// SIMATIC STEP 7 (V5.x) project S7Interface
// CPU: CPU 317-2 PN/DP
// station: Hardware
// station: SIMATIC 300(1)
// station: P_ADR_BUS
// program: Programma S7(1)

SYMBOL_TABLE
"TEST"	DB 1	DB 1
"FETCH"	DB 10	DB 10
"WRITE"	DB 11	DB 11
"FW_TCP"	FB 210	FB 210	// Fetch/Write via TCP
END_SYMBOL_TABLE

// FB 210: know-how protected block, not included

DATA_BLOCK "TEST"	// DB 1
VERSION : 0.1
  STRUCT
   TestBYTE : ARRAY  [0 .. 128 ] OF BYTE ;
   TestCHAR : ARRAY  [0 .. 128 ] OF CHAR ;
   TestWORD : ARRAY  [0 .. 1024 ] OF WORD ;
   TestINT : ARRAY  [0 .. 1024 ] OF INT ;
   TestDWORD : ARRAY  [0 .. 1024 ] OF BOOL ;
   TestDINT : ARRAY  [0 .. 1024 ] OF BOOL ;
   TestBOOL : ARRAY  [0 .. 1024 ] OF BOOL ;
   TestREAL : ARRAY  [0 .. 1024 ] OF REAL ;
   TestSTRING : ARRAY  [0 .. 1024 ] OF STRING  [16 ];
   TestTIME : ARRAY  [0 .. 512 ] OF TIME ;
   TestTOD : ARRAY  [0 .. 512 ] OF TIME_OF_DAY ;
   TestDT : ARRAY  [0 .. 128 ] OF DATE_AND_TIME ;
  END_STRUCT ;	
BEGIN
   TestCHAR[0] := ' ';
   TestCHAR[1] := ' ';
   TestCHAR[2] := ' ';
   TestCHAR[3] := ' ';
   TestCHAR[4] := ' ';
   TestCHAR[5] := ' ';
   TestCHAR[6] := ' ';
   TestCHAR[7] := ' ';
   TestCHAR[8] := ' ';
   TestCHAR[9] := ' ';
   TestCHAR[10] := ' ';
   TestCHAR[11] := ' ';
   TestCHAR[12] := ' ';
   TestCHAR[13] := ' ';
   TestCHAR[14] := ' ';
   TestCHAR[15] := ' ';
   TestCHAR[16] := ' ';
   TestCHAR[17] := ' ';
   TestCHAR[18] := ' ';
   TestCHAR[19] := ' ';
   TestCHAR[20] := ' ';
   TestCHAR[21] := ' ';
   TestCHAR[22] := ' ';
   TestCHAR[23] := ' ';
   TestCHAR[24] := ' ';
   TestCHAR[25] := ' ';
   TestCHAR[26] := ' ';
   TestCHAR[27] := ' ';
   TestCHAR[28] := ' ';
   TestCHAR[29] := ' ';
   TestCHAR[30] := ' ';
   TestCHAR[31] := ' ';
   TestCHAR[32] := ' ';
   TestCHAR[33] := ' ';
   TestCHAR[34] := ' ';
   TestCHAR[35] := ' ';
   TestCHAR[36] := ' ';
   TestCHAR[37] := ' ';
   TestCHAR[38] := ' ';
   TestCHAR[39] := ' ';
   TestCHAR[40] := ' ';
   TestCHAR[41] := ' ';
   TestCHAR[42] := ' ';
   TestCHAR[43] := ' ';
   TestCHAR[44] := ' ';
   TestCHAR[45] := ' ';
   TestCHAR[46] := ' ';
   TestCHAR[47] := ' ';
   TestCHAR[48] := ' ';
   TestCHAR[49] := ' ';
   TestCHAR[50] := ' ';
   TestCHAR[51] := ' ';
   TestCHAR[52] := ' ';
   TestCHAR[53] := ' ';
   TestCHAR[54] := ' ';
   TestCHAR[55] := ' ';
   TestCHAR[56] := ' ';
   TestCHAR[57] := ' ';
   TestCHAR[58] := ' ';
   TestCHAR[59] := ' ';
   TestCHAR[60] := ' ';
   TestCHAR[61] := ' ';
   TestCHAR[62] := ' ';
   TestCHAR[63] := ' ';
   TestCHAR[64] := ' ';
   TestCHAR[65] := ' ';
   TestCHAR[66] := ' ';
   TestCHAR[67] := ' ';
   TestCHAR[68] := ' ';
   TestCHAR[69] := ' ';
   TestCHAR[70] := ' ';
   TestCHAR[71] := ' ';
   TestCHAR[72] := ' ';
   TestCHAR[73] := ' ';
   TestCHAR[74] := ' ';
   TestCHAR[75] := ' ';
   TestCHAR[76] := ' ';
   TestCHAR[77] := ' ';
   TestCHAR[78] := ' ';
   TestCHAR[79] := ' ';
   TestCHAR[80] := ' ';
   TestCHAR[81] := ' ';
   TestCHAR[82] := ' ';
   TestCHAR[83] := ' ';
   TestCHAR[84] := ' ';
   TestCHAR[85] := ' ';
   TestCHAR[86] := ' ';
   TestCHAR[87] := ' ';
   TestCHAR[88] := ' ';
   TestCHAR[89] := ' ';
   TestCHAR[90] := ' ';
   TestCHAR[91] := ' ';
   TestCHAR[92] := ' ';
   TestCHAR[93] := ' ';
   TestCHAR[94] := ' ';
   TestCHAR[95] := ' ';
   TestCHAR[96] := ' ';
   TestCHAR[97] := ' ';
   TestCHAR[98] := ' ';
   TestCHAR[99] := ' ';
   TestCHAR[100] := ' ';
   TestCHAR[101] := ' ';
   TestCHAR[102] := ' ';
   TestCHAR[103] := ' ';
   TestCHAR[104] := ' ';
   TestCHAR[105] := ' ';
   TestCHAR[106] := ' ';
   TestCHAR[107] := ' ';
   TestCHAR[108] := ' ';
   TestCHAR[109] := ' ';
   TestCHAR[110] := ' ';
   TestCHAR[111] := ' ';
   TestCHAR[112] := ' ';
   TestCHAR[113] := ' ';
   TestCHAR[114] := ' ';
   TestCHAR[115] := ' ';
   TestCHAR[116] := ' ';
   TestCHAR[117] := ' ';
   TestCHAR[118] := ' ';
   TestCHAR[119] := ' ';
   TestCHAR[120] := ' ';
   TestCHAR[121] := ' ';
   TestCHAR[122] := ' ';
   TestCHAR[123] := ' ';
   TestCHAR[124] := ' ';
   TestCHAR[125] := ' ';
   TestCHAR[126] := ' ';
   TestCHAR[127] := ' ';
   TestCHAR[128] := ' ';
END_DATA_BLOCK

DATA_BLOCK "FETCH"	// DB 10
TITLE = Connection Parameters for TCON
AUTHOR : SIMATIC
FAMILY : COMM
NAME : TCON_PAR
VERSION : 0.1
  STRUCT
   OUCW_1 : STRUCT
    block_length : WORD  := W#16#40;	//#!FECTH!#
    id : WORD  := W#16#1;
    connection_type : BYTE  := B#16#11;
    active_est : BOOL ;
    local_device_id : BYTE  := B#16#2;
    local_tsap_id_len : BYTE  := B#16#2;
    rem_subnet_id_len : BYTE ;
    rem_staddr_len : BYTE ;
    rem_tsap_id_len : BYTE ;
    next_staddr_len : BYTE ;
    local_tsap_id : ARRAY  [1 .. 16 ] OF BYTE  := B#16#7, B#16#D0, B#16#0, B#16#0, B#16#0, B#16#0, B#16#0, B#16#0, B#16#0, B#16#0, B#16#0, B#16#0, B#16#0, B#16#0, B#16#0, B#16#0;
    rem_subnet_id : ARRAY  [1 .. 6 ] OF BYTE  := B#16#0, B#16#0, B#16#0, B#16#0, B#16#0, B#16#0;
    rem_staddr : ARRAY  [1 .. 6 ] OF BYTE  := B#16#0, B#16#0, B#16#0, B#16#0, B#16#0, B#16#0;
    rem_tsap_id : ARRAY  [1 .. 16 ] OF BYTE  := B#16#0, B#16#0, B#16#0, B#16#0, B#16#0, B#16#0, B#16#0, B#16#0, B#16#0, B#16#0, B#16#0, B#16#0, B#16#0, B#16#0, B#16#0, B#16#0;
    next_staddr : ARRAY  [1 .. 6 ] OF BYTE  := B#16#0, B#16#0, B#16#0, B#16#0, B#16#0, B#16#0;
    spare : WORD ;	//#!FECTH!#
   END_STRUCT ;
  END_STRUCT ;	
BEGIN
   OUCW_1.block_length := W#16#40;
   OUCW_1.id := W#16#1;
   OUCW_1.connection_type := B#16#11;
   OUCW_1.local_device_id := B#16#2;
   OUCW_1.local_tsap_id_len := B#16#2;
   OUCW_1.local_tsap_id[1] := B#16#7;
   OUCW_1.local_tsap_id[2] := B#16#D0;
END_DATA_BLOCK

DATA_BLOCK "WRITE"	// DB 11
TITLE = Connection Parameters for TCON
AUTHOR : SIMATIC
FAMILY : COMM
NAME : TCON_PAR
VERSION : 0.1
  STRUCT
   OUCW_1 : STRUCT
    block_length : WORD  := W#16#40;	//#!WRITE!#
    id : WORD  := W#16#2;
    connection_type : BYTE  := B#16#11;
    active_est : BOOL ;
    local_device_id : BYTE  := B#16#2;
    local_tsap_id_len : BYTE  := B#16#2;
    rem_subnet_id_len : BYTE ;
    rem_staddr_len : BYTE ;
    rem_tsap_id_len : BYTE ;
    next_staddr_len : BYTE ;
    local_tsap_id : ARRAY  [1 .. 16 ] OF BYTE  := B#16#7, B#16#D1, B#16#0, B#16#0, B#16#0, B#16#0, B#16#0, B#16#0, B#16#0, B#16#0, B#16#0, B#16#0, B#16#0, B#16#0, B#16#0, B#16#0;
    rem_subnet_id : ARRAY  [1 .. 6 ] OF BYTE  := B#16#0, B#16#0, B#16#0, B#16#0, B#16#0, B#16#0;
    rem_staddr : ARRAY  [1 .. 6 ] OF BYTE  := B#16#0, B#16#0, B#16#0, B#16#0, B#16#0, B#16#0;
    rem_tsap_id : ARRAY  [1 .. 16 ] OF BYTE  := B#16#0, B#16#0, B#16#0, B#16#0, B#16#0, B#16#0, B#16#0, B#16#0, B#16#0, B#16#0, B#16#0, B#16#0, B#16#0, B#16#0, B#16#0, B#16#0;
    next_staddr : ARRAY  [1 .. 6 ] OF BYTE  := B#16#0, B#16#0, B#16#0, B#16#0, B#16#0, B#16#0;
    spare : WORD ;	//#!WRITE!#
   END_STRUCT ;
  END_STRUCT ;	
BEGIN
   OUCW_1.block_length := W#16#40;
   OUCW_1.id := W#16#2;
   OUCW_1.connection_type := B#16#11;
   OUCW_1.local_device_id := B#16#2;
   OUCW_1.local_tsap_id_len := B#16#2;
   OUCW_1.local_tsap_id[1] := B#16#7;
   OUCW_1.local_tsap_id[2] := B#16#D1;
END_DATA_BLOCK

DATA_BLOCK DB 20
AUTHOR : SIMATIC
FAMILY : COMM
VERSION : 0.0
"FW_TCP"
BEGIN
END_DATA_BLOCK

DATA_BLOCK DB 21
AUTHOR : SIMATIC
FAMILY : COMM
VERSION : 0.0
"FW_TCP"
BEGIN
END_DATA_BLOCK

ORGANIZATION_BLOCK OB 1
TITLE = "Main Program Sweep (Cycle)"
VERSION : 0.1
VAR_TEMP
  OB1_EV_CLASS : BYTE ;	//Bits 0-3 = 1 (Coming event), Bits 4-7 = 1 (Event class 1)
  OB1_SCAN_1 : BYTE ;	//1 (Cold restart scan 1 of OB 1), 3 (Scan 2-n of OB 1)
  OB1_PRIORITY : BYTE ;	//Priority of OB Execution
  OB1_OB_NUMBR : BYTE ;	//1 (Organization block 1, OB1)
  OB1_RESERVED_1 : BYTE ;	//Reserved for system
  OB1_RESERVED_2 : BYTE ;	//Reserved for system
  OB1_PREV_CYCLE : INT ;	//Cycle time of previous OB1 scan (milliseconds)
  OB1_MIN_CYCLE : INT ;	//Minimum cycle time of OB1 (milliseconds)
  OB1_MAX_CYCLE : INT ;	//Maximum cycle time of OB1 (milliseconds)
  OB1_DATE_TIME : DATE_AND_TIME ;	//Date and time OB1 started
END_VAR
BEGIN
NETWORK
TITLE =
      CALL  "FW_TCP" , DB 20 (
           DIX 0.0                  := TRUE,
           DIW 2                    := W#16#1002,
           DIW 4                    := 64,
           DIW 6                    := 10,
           DID 8                    := P#DBX 0.0,
           DIW 12                   := 0,
           DIX 14.0                 := M 0.1,
           DIX 14.1                 := M 0.2,
           DIB 15                   := MB 1,
           DIW 16                   := MW 2);
      CALL  "FW_TCP" , DB 21 (
           DIX 0.0                  := TRUE,
           DIW 2                    := W#16#1002,
           DIW 4                    := 64,
           DIW 6                    := 11,
           DID 8                    := P#DBX 0.0,
           DIW 12                   := 0,
           DIX 14.0                 := M 4.1,
           DIX 14.1                 := M 4.2,
           DIB 15                   := MB 5,
           DIW 16                   := MW 6);
END_ORGANIZATION_BLOCK
